(*

.. <legal notes>

legal notes
=================
| SPDX-FileCopyrightText: © 2026 Oleksandr Tiutyk <trofimich@gmail.com>
| SPDX-License-Identifier: LGPL-3.0-only
| For details check: LGPL-3.0-only_

.. _LGPL-3.0-only: https://www.gnu.org/licenses/lgpl-3.0.en.html

.. </legal notes>

*)

{attribute 'qualified_only'}
VAR_GLOBAL CONSTANT
    POSITIVE_INFINITY_REAL : REAL := TO_REAL(16#7F800000); // IEEE 754 +Infinity
    NEGATIVE_INFINITY_REAL : REAL := TO_REAL(16#FF800000); // IEEE 754 -Infinity
    NAN_REAL : REAL := TO_REAL(16#7FC00000); // IEEE 754 NaN

    POSITIVE_INFINITY_LREAL : LREAL := TO_LREAL(16#7FF0000000000000); // IEEE 754 +Infinity
    NEGATIVE_INFINITY_LREAL : LREAL := TO_LREAL(16#FFF0000000000000); // IEEE 754 -Infinity
    NAN_LREAL : LREAL := TO_LREAL(16#7FF8000000000000); // IEEE 754 NaN
END_VAR

(* stored: Version 1.1.0.1
   GVL Constants: Id {991c0012-6458-465c-8bfe-eea78efbca68} *)
